# EPICS autosave request: iocBoot/ioc13MeasCompE1608_1/auto_settings.req
file "E1608_settings.req", P=13E1608_1:
